TYPE T_JCL_IO :
STRUCT
END_STRUCT
END_TYPE

(* stored: Version 1.1.0.1, ProductVersion 3.1.0.36
   DUT T_JCL_IO: Id {c1bbc3f5-30b2-4961-96b2-30cc6c78adeb} *)
